PROGRAM PRG_CML_03_AdditionalConvCtrl
VAR

END_VAR

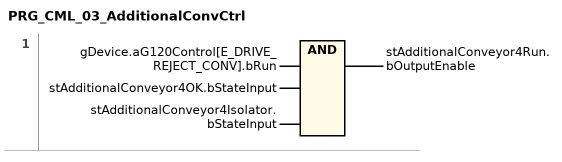
// NETWORK 1
stAdditionalConveyor4Run.bOutputEnable := gDevice.aG120Control[E_DRIVE_REJECT_CONV].bRun AND stAdditionalConveyor4OK.bStateInput AND stAdditionalConveyor4Isolator.bStateInput;

END_PROGRAM

(* stored: Version 1.1.0.1
   POU PRG_CML_03_AdditionalConvCtrl: Id {85f683d5-2a3a-42cb-9844-4397426d4ca2}, SpecialFunc None *)
